FUNCTION_BLOCK FB_HE_SATT_FilterWedge EXTENDS FB_HE_SATT_Filter IMPLEMENTS I_HE_SATT_FilterWedge
VAR
    fThicknessAt0 : LREAL; // 0 is the part of the filter that is the closest to the center of the pipe when retracted.
    fThicknessAtLength : LREAL;
END_VAR


METHOD FB_Init: BOOL
VAR_INPUT
    bInitRetains: BOOL; // TRUE: the retain variables are initialized (reset warm / reset cold)
    bInCopyCode: BOOL;  // TRUE: the instance will be copied to the copy code afterward (online change)   
    
    iHolder : I_HE_SATT_FilterHolder;
    fDefaultLength : LREAL;
    eDefaultMaterial : E_HE_SATT_FilterMaterial;
    eDefaultStatus : E_HE_SATT_FilterStatus;
    fDefaultThicknessAt0 : LREAL;
    fDefaultThicknessAtLength : LREAL;
END_VAR

THIS^.iHolder := iHolder;
THIS^.fLength := fDefaultLength;
THIS^.eMaterial := eDefaultMaterial;
THIS^.eStatus := eDefaultStatus;
THIS^.fThicknessAt0 := fDefaultThicknessAt0;
THIS^.fThicknessAtLength := fDefaultThicknessAtLength;
END_METHOD


PROPERTY MaxThickness : LREAL
GET

MaxThickness := MAX(THIS^.fThicknessAt0, THIS^.fThicknessAtLength);
END_GET
END_PROPERTY


PROPERTY MinThickness : LREAL
GET

MinThickness := MIN(THIS^.fThicknessAt0, THIS^.fThicknessAtLength);
END_GET
END_PROPERTY


METHOD ThicknessAt : LREAL
VAR_INPUT
	(* Position in units of property Length and with value from 0 to value of property Length*)
	fPosition	: LREAL;
END_VAR
END_METHOD

END_FUNCTION_BLOCK

(* stored: Version 1.1.0.1
   POU FB_HE_SATT_FilterWedge: Id {1b346c5d-0a0d-43fc-92fb-3d2a6236cfee}, SpecialFunc None
   Method FB_Init: Id {04a4b23c-2bf7-4e51-be02-82f9b639729e}
   Property MaxThickness: Id {65b1867a-2cd2-46cd-a7f7-861ee80c6273}
   Get Get: Id {442417cc-62b5-49ba-b449-3c53309716c0}
   Property MinThickness: Id {675934c1-6f44-4a35-aa50-d5d7d5b84a48}
   Get Get: Id {c2c8acc4-cb96-42fb-8c29-2b32540fca06}
   Method ThicknessAt: Id {b61cd9fc-b08e-4e7f-9910-87a18d4cffe9} *)
